(* CODESYS project tcdevicebase.library
   Author: ATI Software Engineering
   Version: 2.0.0
   Title: TcDeviceBase
   DefaultNamespace: TcNexa_Devices_Base_TcDeviceBase
   Placeholder: TcDeviceBase
   Company: TcNexa

Project tree, tasks and I/O mapping:
  libraries: Tc2_Standard, * (Beckhoff Automation GmbH); Tc2_System, * (Beckhoff Automation GmbH); Tc3_IotBase, * (Beckhoff Automation GmbH); Tc3_Module, * (Beckhoff Automation GmbH); TcNexaHmi, * (TcNexa); TcProcess, * (TcNexa); TcUtilities, * (TcNexa)
  Base/
    DUTs/
      data type ST_MethodState
    POUs/
      function block FB_DeviceBase [ST]: methodTimeout, _getBusyMessage, _getErrorMessage, _methodFooter, _methodHeader, FB_init, FB_main
      function block FB_DeviceNexaHmi [ST]: _handleMessageQueue, _init, _onConnection, FB_init, cellTag, deviceName, deviceTag, hostName, hostPort, isConnected, messageFullTopic, messageLastTopicLevel, messagePayload, onNewMessage, stationTag, topicPrefix, FB_main, publish, publishAdr, subscribe, unsubscribe
  Components/
    function block FB_DeviceButtonNexaHmi [ST]: _handleNewMessages, _onConnection, _updateTopics, FB_init, enabled, focused, loggingEnabled, name, onLongPress, onTap, onTapDown, onTapUp, FB_main
  Tests/
    program PRG_TEST [ST]
  Version/
    global variables Global_Version
*)

// Base/DUTs/ST_MethodState
TYPE ST_MethodState :
STRUCT
	init		: BOOL;
	execute		: BOOL;
	timeout		: BOOL;
END_STRUCT
END_TYPE

// Version/Global_Version
{attribute 'TcGenerated'}
{attribute 'no-analysis'}
{attribute 'linkalways'}
// This function has been automatically generated from the project information.
VAR_GLOBAL CONSTANT
	{attribute 'const_non_replaced'}
	stLibVersion_TcDeviceBase : ST_LibVersion := (iMajor := 2, iMinor := 0, iBuild := 0, iRevision := 0, nFlags := 0, sVersion := '2.0.0');
END_VAR

// Base/POUs/FB_DeviceBase
FUNCTION_BLOCK ABSTRACT FB_DeviceBase
VAR
	_Step					: TcNexa_Components_TcProcess.FB_Step;
	_InternalResponse		: TcNexa_Components_TcProcess.FB_MethodResponse;
	_calledMethod			: STRING;
	_tmpText				: Tc2_System.T_MaxString;
	_methodTimeout			: Tc2_Standard.TON;
	_methodState			: ST_MethodState;
	_executeMethod			: BOOL;
	_name					: STRING;
	_tag					: STRING;
	_nameTag				: STRING;
	_methodTime				: TIME:= T#5S;
	_noMethodCalledTrigger	: Tc2_Standard.R_TRIG;
END_VAR

PROPERTY methodTimeout : TIME
GET
methodTimeout:= _methodTime;
END_GET
SET
_methodTime:= methodTimeout;
END_SET
END_PROPERTY

METHOD PROTECTED _getBusyMessage : STRING(255)
VAR_INPUT
	message		: STRING(255);
END_VAR
_getBusyMessage:= Tc2_Standard.CONCAT(STR1:= _nameTag, STR2:= ' ');
_getBusyMessage:= Tc2_Standard.CONCAT(STR1:= _getBusyMessage, STR2:= _calledMethod);
_getBusyMessage:= Tc2_Standard.CONCAT(STR1:= _getBusyMessage, STR2:= ' ');
_getBusyMessage:= Tc2_Standard.CONCAT(STR1:= _getBusyMessage, STR2:= message);
END_METHOD

METHOD PROTECTED _getErrorMessage : STRING(255)
VAR_INPUT
END_VAR
_getErrorMessage:= Tc2_Standard.CONCAT(STR1:= _nameTag, STR2:= ' failed during ');
_getErrorMessage:= Tc2_Standard.CONCAT(STR1:= _getErrorMessage, STR2:= _calledMethod);
END_METHOD

METHOD PROTECTED _methodFooter
VAR_INPUT
	Response		: REFERENCE TO TcNexa_Components_TcProcess.FB_MethodResponse;
END_VAR
IF NOT _InternalResponse.busy THEN _calledMethod:= ''; END_IF
IF __ISVALIDREF(Response) THEN Response.copyFrom(Response:= _InternalResponse); END_IF
END_METHOD

METHOD PROTECTED _methodHeader : ST_MethodState
VAR_INPUT
	methodName		: Tc2_System.T_MaxString;
END_VAR
IF (_calledMethod = '') THEN
	_calledMethod:= methodName;
	_Step.init();
	_methodTimeout(IN:= FALSE);
	_methodHeader.init:= TRUE;
	_methodHeader.execute:= TRUE;
	_executeMethod:= TRUE;
	_InternalResponse.setBusy(message:= methodName);
ELSIF (_calledMethod = methodName) THEN
	_executeMethod:= TRUE;
	_methodTimeout(IN:= TRUE, PT:= _methodTime);
	IF _methodTimeout.Q THEN
		_InternalResponse.setFail(message:= _getErrorMessage(), description:= 'Timeout occurred');
		_methodHeader.timeout:= TRUE;
	ELSE
		_InternalResponse.setBusy(message:= _getBusyMessage(message:= 'in progress'));
		_methodHeader.execute:= TRUE;
	END_IF
ELSE
	_InternalResponse.setBusy(message:= _getBusyMessage(message:= 'in progress'));
END_IF
END_METHOD

METHOD FB_init : BOOL
VAR_INPUT
	bInitRetains 	: BOOL; // if TRUE, the retain variables are initialized (warm start / cold start)
	bInCopyCode 	: BOOL;  // if TRUE, the instance afterwards gets moved into the copy code (online change)
	name			: STRING;
	tag				: STRING;
END_VAR
THIS^._name:= name;
THIS^._tag:= tag;

IF (name = '') THEN
	_nameTag:= tag;
ELSE
	_nameTag:= name;
	IF (_tag <> '') THEN
		_nameTag:= Tc2_Standard.CONCAT(STR1:= _nameTag, STR2:= ' (');
		_nameTag:= Tc2_Standard.CONCAT(STR1:= _nameTag, STR2:= tag);
		_nameTag:= Tc2_Standard.CONCAT(STR1:= _nameTag, STR2:= ')');
	END_IF
END_IF
END_METHOD

METHOD PUBLIC FB_main
VAR_INPUT
END_VAR
_noMethodCalledTrigger(CLK:= (_calledMethod = ''));

IF (_calledMethod <> '') AND NOT _executeMethod THEN
	_calledMethod:= '';
END_IF

_executeMethod:= FALSE;
END_METHOD

END_FUNCTION_BLOCK

// Base/POUs/FB_DeviceNexaHmi
FUNCTION_BLOCK FB_DeviceNexaHmi IMPLEMENTS TcNexa_Devices_Hmi_TcNexaHmi.I_NexaHmi
VAR
	(* Mqtt *)
	_Client						: Tc3_IotBase.FB_IotMqttClient;
	_ClientMessageQueue			: Tc3_IotBase.FB_IotMqttMessageQueue;
	_ClientMessage				: Tc3_IotBase.FB_IotMqttMessage;
	_isInit						: BOOL;
	_onClientConnection			: Tc2_Standard.R_TRIG;
	_isClientConnected			: BOOL;
	_onNewMessage				: BOOL;
	_willPayload				: STRING;
	_topicPrefix				: STRING(255);
	(* Message *)
	_messageTopic				: Tc2_System.T_MaxString;
	_messageLastTopicLevel		: Tc2_System.T_MaxString;
	_messageTopicSplitter		: TcNexa_Components_TcUtilities.FB_TextSplitter;
	_messagePayload				: Tc2_System.T_MaxString;		
	(* General *)
	_timerPublish				: Tc2_Standard.TON;		
	_tmpText					: Tc2_System.T_MaxString;					
	_tmpCounter					: USINT;			
	(* Information *)
	_cellTag					: STRING;
	_stationTag					: STRING;
	_tag						: STRING;
	_name						: STRING;
	_deviceType					: STRING;
END_VAR

METHOD PROTECTED _handleMessageQueue
VAR_INPUT
END_VAR
_onNewMessage:= FALSE;
IF (_ClientMessageQueue.nQueuedMessages > 0) THEN
	IF _ClientMessageQueue.Dequeue(fbMessage:= _ClientMessage)  THEN
		_ClientMessage.GetTopic(
			pTopic				:= ADR(_messageTopic),
			nTopicSize			:= SIZEOF(_messageTopic));
		_ClientMessage.GetPayload(
			pPayload			:= ADR(_messagePayload),
			nPayloadSize		:= SIZEOF(_messagePayload),
			bSetNullTermination	:= TRUE);
		_messageTopicSplitter.split(
			source				:= _messageTopic,
			delimiter			:= '/',
			Response			:= 0);
		_messageLastTopicLevel:= _messageTopicSplitter.getValueAt(
			index				:= _messageTopicSplitter.size,
			Response			:= 0);
		_onNewMessage:= TRUE;
	END_IF
ELSE
	_messageTopic:= '';
	_messagePayload:= '';
END_IF
END_METHOD

METHOD PROTECTED _init
VAR_INPUT
END_VAR
IF _isInit THEN RETURN; END_IF
_isInit:= TRUE;

_Client.ipMessageQueue:= _ClientMessageQueue;

_tmpText:= '';
IF (_cellTag <> '') THEN
	_tmpText:= Tc2_Standard.CONCAT(STR1:= _cellTag, STR2:= '/');
END_IF
IF (_stationTag <> '') THEN
	_tmpText:= Tc2_Standard.CONCAT(STR1:= _tmpText, STR2:= _stationTag);
	_tmpText:= Tc2_Standard.CONCAT(STR1:= _tmpText, STR2:= '/');
END_IF
//_tmpText:= Tc2_Standard.CONCAT(STR1:= _tmpText, STR2:= 'devices/');
//_tmpText:= Tc2_Standard.CONCAT(STR1:= _tmpText, STR2:= _deviceType);
//_tmpText:= Tc2_Standard.CONCAT(STR1:= _tmpText, STR2:= '/');
//_tmpText:= Tc2_Standard.CONCAT(STR1:= _tmpText, STR2:= _tag);
//_tmpText:= Tc2_Standard.CONCAT(STR1:= _tmpText, STR2:= '/');
_topicPrefix:= '';
_topicPrefix:= Tc2_Standard.CONCAT(STR1:= _topicPrefix, STR2:= 'devices/');
_topicPrefix:= Tc2_Standard.CONCAT(STR1:= _topicPrefix, STR2:= _deviceType);
_topicPrefix:= Tc2_Standard.CONCAT(STR1:= _topicPrefix, STR2:= '/');
_topicPrefix:= Tc2_Standard.CONCAT(STR1:= _topicPrefix, STR2:= _tag);
_topicPrefix:= Tc2_Standard.CONCAT(STR1:= _topicPrefix, STR2:= '/');

_Client.sTopicPrefix:= _tmpText;
_Client.sClientId:= CONCAT(STR1:= _tmpText, STR2:= _topicPrefix);
(* Will *)
_willPayload:= BOOL_TO_STRING(FALSE);
_Client.stWill.sTopic:= Tc2_Standard.CONCAT(STR1:= _topicPrefix, STR2:= 'active');
_Client.stWill.pPayload:= ADR(_willPayload);
_Client.stWill.nPayloadSize:= INT_TO_UDINT(Tc2_Standard.LEN(_willPayload));
_Client.stWill.eQoS:= TcIotMqttQos.AtMostOnceDelivery;
_Client.stWill.bRetain:= TRUE;
END_METHOD

METHOD PROTECTED _onConnection
VAR_INPUT
END_VAR
IF NOT _onClientConnection.Q THEN RETURN; END_IF

(*** PUBLISH ***)
publish(
	topic	:= 'active',
	payload	:= BOOL_TO_STRING(TRUE));
publish(
	topic	:= 'general/name',
	payload	:= _name);
END_METHOD

METHOD FB_init : BOOL
VAR_INPUT
	bInitRetains 	: BOOL; 	// if TRUE, the retain variables are initialized (warm start / cold start)
	bInCopyCode 	: BOOL;  	// if TRUE, the instance afterwards gets moved into the copy code (online change)
	deviceType		: STRING;
END_VAR
THIS^._deviceType:= deviceType;
END_METHOD

PROPERTY cellTag : STRING
GET
cellTag:= _cellTag;
END_GET
SET
_cellTag:= cellTag;
END_SET
END_PROPERTY

PROPERTY deviceName : STRING
GET
deviceName:= _name;
END_GET
SET
_name:= deviceName;
END_SET
END_PROPERTY

PROPERTY deviceTag : STRING
GET
deviceTag:= _tag;
END_GET
SET
_tag:= deviceTag;
END_SET
END_PROPERTY

PROPERTY PUBLIC hostName : Tc2_System.T_MaxString
GET
hostName:= _Client.sHostName;
END_GET
SET
_Client.sHostName:= hostName;
END_SET
END_PROPERTY

PROPERTY PUBLIC hostPort : UINT
GET
hostPort:= _Client.nHostPort;
END_GET
SET
_Client.nHostPort:= hostPort;
END_SET
END_PROPERTY

PROPERTY PUBLIC isConnected : BOOL
GET
isConnected:= _Client.bConnected;
END_GET
END_PROPERTY

PROPERTY messageFullTopic : Tc2_System.T_MaxString
GET
messageFullTopic:= _messageTopic;
END_GET
END_PROPERTY

PROPERTY PUBLIC messageLastTopicLevel : STRING
GET
messageLastTopicLevel:= _messageLastTopicLevel;
END_GET
END_PROPERTY

PROPERTY messagePayload : Tc2_System.T_MaxString
GET
messagePayload:= _messagePayload;
END_GET
END_PROPERTY

PROPERTY PUBLIC onNewMessage : BOOL
GET
onNewMessage:= _onNewMessage;
END_GET
END_PROPERTY

PROPERTY stationTag : STRING
GET
stationTag:= _stationTag;
END_GET
SET
_stationTag:= stationTag;
END_SET
END_PROPERTY

PROPERTY PUBLIC topicPrefix : Tc2_System.T_MaxString
GET
topicPrefix:= _Client.sClientId;//_Client.sTopicPrefix;
END_GET
END_PROPERTY

METHOD PUBLIC FB_main
VAR_INPUT
END_VAR
_init();

_Client.Execute(bConnect:= TRUE);
_isClientConnected:= _Client.bConnected;
_onClientConnection(CLK:= _isClientConnected);

_onConnection();
_handleMessageQueue();
END_METHOD

METHOD PUBLIC publish : BOOL
VAR_INPUT
	topic		: Tc2_System.T_MaxString;
	payload		: Tc2_System.T_MaxString;
END_VAR
_tmpText:= Tc2_Standard.CONCAT(
	STR1:= _topicPrefix,
	STR2:= topic);

publish:= _Client.Publish(
			sTopic			:= _tmpText,
			pPayload		:= ADR(payload),
			nPayloadSize	:= INT_TO_UDINT(Tc2_Standard.LEN(payload)),
			eQoS			:= TcIotMqttQos.AtMostOnceDelivery,
			bRetain			:= TRUE,
			bQueue			:= FALSE);
END_METHOD

METHOD PUBLIC publishAdr : BOOL
VAR_INPUT
	topic		: Tc2_System.T_MaxString;
	payload		: PVOID;
	payloadSize	: UDINT;
END_VAR
_tmpText:= Tc2_Standard.CONCAT(
	STR1:= _topicPrefix,
	STR2:= topic);

publishAdr:= _Client.Publish(
			sTopic			:= _tmpText,
			pPayload		:= payload,
			nPayloadSize	:= payloadSize,
			eQoS			:= TcIotMqttQos.AtMostOnceDelivery,
			bRetain			:= TRUE,
			bQueue			:= FALSE);
END_METHOD

METHOD PUBLIC subscribe : BOOL
VAR_INPUT
	topic		: Tc2_System.T_MaxString;
END_VAR
_tmpText:= Tc2_Standard.CONCAT(
	STR1:= _topicPrefix,
	STR2:= topic);

subscribe:= _Client.Subscribe(
				sTopic	:= _tmpText,
				eQoS	:= TcIotMqttQos.AtLeastOnceDelivery);
END_METHOD

METHOD PUBLIC unsubscribe
VAR_INPUT
	topic		: Tc2_System.T_MaxString;
END_VAR
_tmpText:= Tc2_Standard.CONCAT(
	STR1:= _topicPrefix,
	STR2:= topic);

_Client.Unsubscribe(sTopic:= _tmpText);
END_METHOD

END_FUNCTION_BLOCK

// Components/FB_DeviceButtonNexaHmi
FUNCTION_BLOCK FB_DeviceButtonNexaHmi
VAR
	_Hmi					: TcNexa_Devices_Hmi_TcNexaHmi.I_NexaHmi;
	_onHmiConnection		: Tc2_Standard.R_TRIG;
	_isHmiConnected			: BOOL;
	_topicPrefix			: Tc2_System.T_MaxString;
	_topic					: Tc2_System.T_MaxString;
	_tmpText				: Tc2_System.T_MaxString;
	_name					: STRING;
	_enabled				: BOOL;
	_focused				: BOOL;
	_onTap					: BOOL;
	_onTapDown				: BOOL;
	_onTapUp				: BOOL;
	_onLongPress			: BOOL;
	(* *)               	
	_lastName				: STRING;
	_lastEnabled			: BOOL;
	_lastFocused			: BOOL;
	_loggingEnabled			: BOOL;
	_lastLoggingEnabled		: BOOL;
END_VAR

METHOD PROTECTED _handleNewMessages
VAR_INPUT
END_VAR
_onTap:= FALSE;
_onTapDown:= FALSE;
_onTapUp:= FALSE;
_onLongPress:= FALSE;

IF NOT _isHmiConnected THEN RETURN; END_IF

IF _Hmi.onNewMessage THEN
	_tmpText:= Tc2_Standard.CONCAT(STR1:= _Hmi.topicPrefix, STR2:= _topicPrefix);
	IF (_Hmi.messageFullTopic = Tc2_Standard.CONCAT(STR1:= _tmpText, STR2:= 'action')) THEN
		IF (_Hmi.messagePayload = 'tap') AND _enabled THEN
			_onTap:= TRUE;
		ELSIF  (_Hmi.messagePayload = 'tapDown') AND _enabled THEN
			_onTapDown:= TRUE;
		ELSIF  (_Hmi.messagePayload = 'tapUp') AND _enabled THEN
			_onTapUp:= TRUE;
		ELSIF  (_Hmi.messagePayload = 'onLongPress') AND _enabled THEN
			_onLongPress:= TRUE;
		END_IF
	END_IF
END_IF
END_METHOD

METHOD PROTECTED _onConnection
VAR_INPUT
END_VAR
IF NOT _onHmiConnection.Q THEN RETURN; END_IF

IF (Tc2_Standard.RIGHT(STR:= _topic, SIZE:= 1) <> '/') THEN
	_topicPrefix:= Tc2_Standard.CONCAT(STR1:= _topic, STR2:= '/');
ELSE
	_topicPrefix:= _topic;
END_IF
_Hmi.subscribe(topic:= CONCAT(STR1:= _topicPrefix, STR2:= 'action'));
END_METHOD

METHOD PROTECTED _updateTopics
VAR_INPUT
END_VAR
IF NOT _isHmiConnected THEN RETURN; END_IF

(* Name *)
IF (_lastName <> _name) OR _onHmiConnection.Q THEN
	_lastName:= _name;
	_Hmi.publish(
		topic	:= Tc2_Standard.CONCAT(STR1:= _topicPrefix, STR2:= 'name'),
		payload	:= _name);
END_IF
(* Enabled *)
IF (_lastEnabled <> _enabled) OR _onHmiConnection.Q THEN
	_lastEnabled:= _enabled;
	_Hmi.publish(
		topic	:= Tc2_Standard.CONCAT(STR1:= _topicPrefix, STR2:= 'enabled'),
		payload	:= BOOL_TO_STRING(_enabled));
END_IF
(* Focused *)
IF (_lastFocused <> _focused) OR _onHmiConnection.Q THEN
	_lastFocused:= _focused;
	_Hmi.publish(
		topic	:= Tc2_Standard.CONCAT(STR1:= _topicPrefix, STR2:= 'focused'),
		payload	:= BOOL_TO_STRING(_focused));
END_IF
(* Logging Enabled *)
IF (_lastLoggingEnabled <> _loggingEnabled) OR _onHmiConnection.Q THEN
	_lastLoggingEnabled:= _loggingEnabled;
	_Hmi.publish(
		topic	:= Tc2_Standard.CONCAT(STR1:= _topicPrefix, STR2:= 'loggingEnabled'),
		payload	:= BOOL_TO_STRING(_loggingEnabled));
END_IF
END_METHOD

METHOD FB_init : BOOL
VAR_INPUT
	bInitRetains	: BOOL; // if TRUE, the retain variables are initialized (warm start / cold start)
	bInCopyCode 	: BOOL;  // if TRUE, the instance afterwards gets moved into the copy code (online change)
	Hmi				: I_NexaHmi;
	topic			: Tc2_System.T_MaxString;
END_VAR
THIS^._Hmi:= Hmi;
THIS^._topic:= topic;
END_METHOD

PROPERTY enabled : BOOL
GET
enabled:= _enabled;
END_GET
SET
_enabled:= enabled;
END_SET
END_PROPERTY

PROPERTY focused : BOOL
GET
focused:= _focused;
END_GET
SET
_focused:= focused;
END_SET
END_PROPERTY

PROPERTY loggingEnabled : BOOL
GET
loggingEnabled:= _loggingEnabled;
END_GET
SET
_loggingEnabled:= loggingEnabled;
END_SET
END_PROPERTY

PROPERTY PUBLIC name : STRING
GET
name:= _name;
END_GET
SET
_name:= name;
END_SET
END_PROPERTY

PROPERTY onLongPress : BOOL
GET
onLongPress:= _onLongPress;
END_GET
END_PROPERTY

PROPERTY onTap : BOOL
GET
onTap:= _onTap;
END_GET
END_PROPERTY

PROPERTY onTapDown : BOOL
GET
onTapDown:= _onTapDown;
END_GET
END_PROPERTY

PROPERTY onTapUp : BOOL
GET
onTapUp:= _onTapUp;
END_GET
END_PROPERTY

METHOD PUBLIC FB_main
VAR_INPUT
END_VAR
_isHmiConnected:= _Hmi.isConnected;
_onHmiConnection(CLK:= _isHmiConnected);

_onConnection();
_updateTopics();
_handleNewMessages();
END_METHOD

END_FUNCTION_BLOCK

// Tests/PRG_TEST
PROGRAM PRG_TEST
VAR
	_test : FB_DeviceBase;
	_test1	: FB_DeviceNexaHmi;
END_VAR

END_PROGRAM
